// TwinCAT 3 PLC project PLCSim
// ProgramVersion: 3.1.4024.0
// libraries:
//   Tc2_Standard, * (Beckhoff Automation GmbH)
//   Tc2_System, * (Beckhoff Automation GmbH)
//   Tc3_Module, * (Beckhoff Automation GmbH)
// project tree:
//   / GlobalTextList.TcGTLO, PlcTask.TcTTO, Visualization Manager.TcVMO (not stored)
//   GVLs/ GVL.TcGVL
//   POUs/ MAIN.TcPOU, Motor_Control.TcPOU, Process.TcPOU
//   VISUs/ Visualization.TcVIS
// real-time tasks:
//   TASK PlcTask: cycle T#10ms, priority 20, ADS port 350
//   TASK PlcTask1: cycle T#10ms, priority 21, ADS port 351
// variable links:
//   PLCSim/PLCSim Instance <-> PLCStudent/PLCStudent Instance
//     PlcTask Inputs/GVL.ixGotoPosA <-> PlcTask Outputs/GVL.qxGotoPosA
//     PlcTask Inputs/GVL.ixGotoPosB <-> PlcTask Outputs/GVL.qxGotoPosB
//     PlcTask Outputs/GVL.qxA <-> PlcTask Inputs/GVL.ixA
//     PlcTask Outputs/GVL.qxB <-> PlcTask Inputs/GVL.ixB
//     PlcTask Outputs/GVL.qxTram <-> PlcTask Inputs/GVL.ixTram

CONFIGURATION PLCSim
    RESOURCE PLC ON TwinCAT3
        TASK PlcTask(INTERVAL := T#10ms, PRIORITY := 20);
        PROGRAM MAIN WITH PlcTask : MAIN;
    END_RESOURCE
END_CONFIGURATION

// ---- GVLs/GVL.TcGVL
{attribute 'qualified_only'}
VAR_GLOBAL
	//Output from process
	qxTram	AT %Q*: BOOL;
	qxA		AT %Q*: BOOL;
	qxB		AT %Q*: BOOL;
	
	//Input to from Operator
	ixGotoPosB AT %I*: BOOL;
	ixGotoPosA AT %I*: BOOL;
	//icStop AT %I*: BOOL;
	//ixEmergency AT %I*: BOOL;
END_VAR

// ---- POUs/MAIN.TcPOU
PROGRAM MAIN
VAR
END_VAR

Motor_Control();

END_PROGRAM

// ---- POUs/Motor_Control.TcPOU
PROGRAM Motor_Control
VAR
	Process_0: Process;
	Pos: INT;
END_VAR

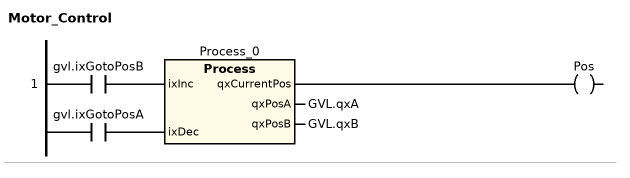
// NETWORK 1
Process_0(ixInc := gvl.ixGotoPosB, ixDec := gvl.ixGotoPosA, qxPosA => GVL.qxA, qxPosB => GVL.qxB); // Process
Pos := Process_0.qxCurrentPos;

END_PROGRAM

// ---- POUs/Process.TcPOU
FUNCTION_BLOCK Process
VAR_INPUT
	ixInc:BOOL;
	ixDec:BOOL;
END_VAR
VAR_OUTPUT
	qxCurrentPos:INT;
	qxPosA:BOOL;
	qxPosB:BOOL;
END_VAR
VAR
END_VAR

IF ixInc AND qxCurrentPos<486 THEN
	qxCurrentPos:= qxCurrentPos + 1;
ELSIF ixDec AND qxCurrentPos>0 THEN
	qxCurrentPos:= qxCurrentPos - 1;
END_IF

IF qxCurrentPos = 486 THEN
	qxPosB:= TRUE;
ELSIF qxCurrentPos = 0 THEN
	qxPosA:= TRUE;
ELSE
	qxPosB:= FALSE;
	qxPosA:= FALSE;
END_IF

END_FUNCTION_BLOCK

// ---- GlobalTextList.TcGTLO
TEXTLIST GlobalTextList
  635 = 'A'
  404 = 'B'
  836 = 'Sa'
  339 = 'Sb'
  850 = 'Train'
END_TEXTLIST

// ---- VISUs/Visualization.TcVIS
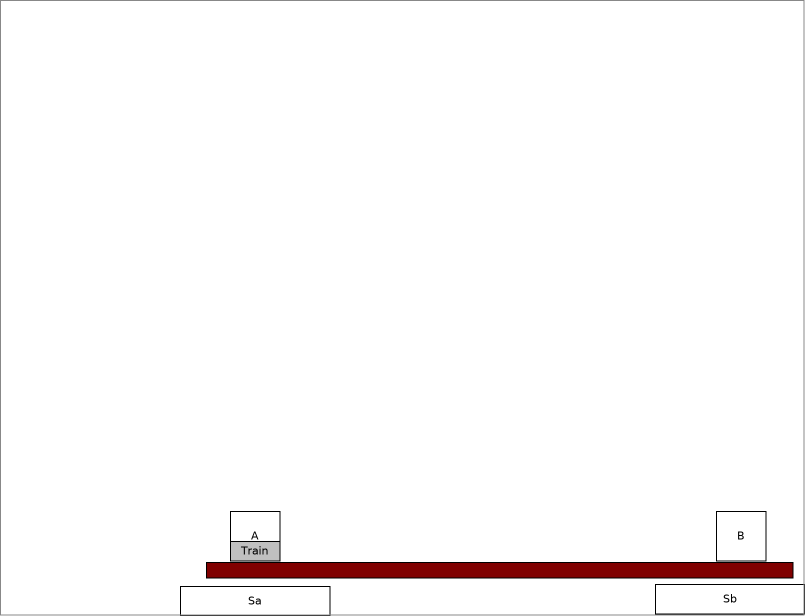
VISUALIZATION Visualization  // 805x616
    Rectangle (206,562 587x16)
    Rectangle (230,511 50x50), "A"
    Rectangle (716,511 50x50), "B"
    Rectangle (230,541 50x20), "Train"
        p3560616238: Motor_Control.Pos
    Rectangle (180,586 150x30), "Sa", colour toggle: GVL.qxA
    Rectangle (655,584 150x30), "Sb", colour toggle: GVL.qxB
END_VISUALIZATION
